SUBAPPLICATION Uebung_007 (* Subapplication Type *)
  (* Standard: 61499-2 *)
  (* Version 1.0, 2023-10-23, franz *)
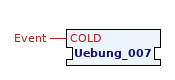
  EVENT_INPUT
    COLD;
  END_EVENT
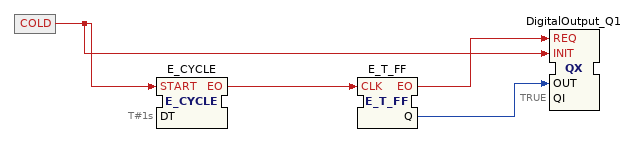
  FBS
    DigitalOutput_Q1 : QX(QI := TRUE);
    E_CYCLE : E_CYCLE(DT := T#1s);
    E_T_FF : E_T_FF;
  END_FBS
  EVENT_CONNECTIONS
    E_CYCLE.EO TO E_T_FF.CLK;
    E_T_FF.EO TO DigitalOutput_Q1.REQ;
    COLD TO DigitalOutput_Q1.INIT;
    COLD TO E_CYCLE.START;
  END_CONNECTIONS
  DATA_CONNECTIONS
    E_T_FF.Q TO DigitalOutput_Q1.OUT;
  END_CONNECTIONS
END_SUBAPPLICATION
